FUNCTION_BLOCK FB_BronkhorstMFM
VAR_INPUT
END_VAR
VAR_OUTPUT
END_VAR
VAR
        {attribute 'pytmc' := '
            pv:
         '}
        stMFM	:	ST_BhElFlow;
END_VAR

//stMFM.i_rFlow = Output;

END_FUNCTION_BLOCK

(* stored: Version 1.1.0.1, ProductVersion 3.1.4022.18
   POU FB_BronkhorstMFM: Id {6583b79d-8f50-416f-b9a8-da0bf6f716a8}, SpecialFunc None *)
